Yaskawa INFORM job: GETPOS.JBI

/JOB
//NAME GETPOS
//POS
///NPOS 0,0,0,0,0,0
//INST
///DATE 2014/10/01 08:55
///ATTR SC,RW,MC
///GROUP1 RB1,BS1
///LVARS 6,0,0,0,0,1,0,0
NOP
GETARG LB000 IARG#(1)
SET LB001 0
SET LB002 3
SKILLSND "LGETPOS LT:0 B0:1 B1:2"
GETARG LB004 IARG#(2)
GETARG LB005 IARG#(3)
SET P[LB004] LP000
SET B[LB005] LB003
END
